FUNCTION_BLOCK POS_SENSE (* Workpiece position sensor *)
  (* Standard: 61499-1; Classification: Simulation *)
  (* Version 0.1, 2005-06-01, JHC, Holobloc Inc, Recompiled with new emitter. *)
  (* Version 0.0, 2004-09-21, JHC, Rockwell Automation *)
  (* Compiler header: package fb.rt.mva; *)
  (* Compiler Java Sun JDK 1.4.2 *)
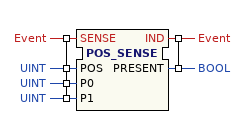
  EVENT_INPUT
    SENSE WITH POS, P0, P1; (* Input change notification *)
  END_EVENT
  EVENT_OUTPUT
    IND WITH PRESENT; (* Output change indication *)
  END_EVENT
  VAR_INPUT
    POS : UINT; (* Workpiece position on conveyor (0-100%) *)
    P0 : UINT; (* Position sensor lower limit *)
    P1 : UINT; (* Position sensor upper limit *)
  END_VAR
  VAR_OUTPUT
    PRESENT : BOOL; (* Workpiece is present between P0 and P1 *)
  END_VAR
  ALGORITHM SENSE IN Java:
boolean newpres = (POS.value>=P0.value) & (POS.value<=P1.value);
if(newpres!=PRESENT.value){
   PRESENT.value = newpres;
   IND.serviceEvent(this);}
  END_ALGORITHM
END_FUNCTION_BLOCK
